# EPICS autosave request: iocBoot/generic_motors_ioc/dbSave/WS_Av_.req
%
% BURT Request File
%
% $(P)WS:Av:  White beam slits, Vertical Aperture
%

file assy.req ASSY=$(P)WS:Av
$(P)WS:Av:Invert
file mtr1.req MTR1=$(P)WS:mt
file mtr1.req MTR1=$(P)WS:mb
file drv1.req DRV1=$(P)WS:ZT
file drv1.req DRV1=$(P)WS:ZB
file axs1.req AXS1=$(P)WS:ZC
file axs1.req AXS1=$(P)WS:ZS
